// TwinCAT 3 PLC project MyPLC
// ProgramVersion: 3.1.4022.0
// libraries:
//   Tc2_Standard, * (Beckhoff Automation GmbH)
//   Tc2_System, * (Beckhoff Automation GmbH)
//   Tc2_Utilities, * (Beckhoff Automation GmbH)
//   Tc3_Module, * (Beckhoff Automation GmbH)
// project tree:
//   DUTs/Error Monitoring/ ST_HRErrHist.TcDUT
//   DUTs/Signal Generator/ E_DistributionType.TcDUT, E_FunctionType.TcDUT
//   GVLs/ GVL_Constant.TcGVL, GVL_LabviewDataShare.TcGVL
//   / PlcTask.TcTTO
//   POUs/Error Monitoring/ FB_HRErrHist.TcPOU
//   POUs/Signal Generator/ FB_FunctionGenerator.TcPOU (not stored), FB_NoiseGenerator.TcPOU
//   POUs/ MAIN.TcPOU
// real-time tasks:
//   TASK GetDataTask: cycle T#5ms, priority 6, ADS port 350

CONFIGURATION MyPLC
    RESOURCE PLC ON TwinCAT3
        TASK PlcTask(INTERVAL := T#5ms, PRIORITY := 6);
        PROGRAM MAIN WITH PlcTask : MAIN;
    END_RESOURCE
END_CONFIGURATION

// ---- DUTs/Error Monitoring/ST_HRErrHist.TcDUT
TYPE ST_HRErrHist :
STRUCT
{attribute 'displaymode':='hex'}
	hrErrCode	: HRESULT;
	sErrSource	: STRING(63);
	nErrCount	: UDINT;
END_STRUCT
END_TYPE

// ---- DUTs/Signal Generator/E_DistributionType.TcDUT
{attribute 'qualified_only'}
TYPE E_DistributionType :
(
	Uniform := 0,
	Normal,
	Chi_squared,
	Exponential,
	Gamma
);
END_TYPE

// ---- DUTs/Signal Generator/E_FunctionType.TcDUT
{attribute 'qualified_only'}
TYPE E_FunctionType :
(
	Sine,		// typical for vibrations originating from rotating machine
	Square,		// mixed sine signals good for analyzing spectrum
	Pulse,		// mixed sine signals good for analyzing spectrum
	Triangular,	// mixed sine signals good for analyzing spectrum
	Sawtooth,	// ramp-type vibrations, continuously increasing
	AM			// amplitude modulation: typical for vibrations originating from gear-tooth failure or bearing faults
);
END_TYPE

// ---- GVLs/GVL_Constant.TcGVL
VAR_GLOBAL CONSTANT
	
	// input definition
	cChannels		: UDINT 	:= 4;    // number of input channels
	cOversamples 	: UDINT 	:= 10;	 // oversamples from input terminal
	
	// pupulation for statistical calculations
	cPupulation 	: UDINT     := 6000;	
	
	// Source MultiArray
	cBufferLength : UDINT := 100; 
	
	// wait for cAppendData MultiArrays with cBufferLength Elements before calculating | Elements in total = cPupulation 
	cAppendData     : UDINT := cPupulation/cBufferLength;
	
END_VAR

// ---- GVLs/GVL_LabviewDataShare.TcGVL
{attribute 'qualified_only'}
VAR_GLOBAL
	
	//Cal Station Variables	
	out_bInitializeStartupRoutine : BOOL;
	
	 // Beckhoff to Labview MQTT Info Transfer - Current Sensor DeviceID
    out_strDeviceID_labview : STRING;

    // Beckhoff to Labview MQTT Info Transfer - Current Lot running on the Machine
    out_strLotNo_labview : STRING;

    // Beckhoff to Labview MQTT Info Transfer - 1) Calibration 2) FFT
    out_strTestMode_labview : STRING;

    // Beckhoff to Labview MQTT Info Transfer - Interrupt Signal from Beckhoff to Labview to Abort the Calibration Process
    out_bAbortCalibrationSequence_labview : BOOL;

    // Beckhoff to Labview MQTT Info Transfer - Boolean to Indicate if the current sequence are for Master Parts or not
    out_bMasterSequenceActive_labview : BOOL;

    // Beckhoff to Labview MQTT Info Transfer - Boolean indicating the Beckhoff is Active
    out_bBeckhoffHandshakeBit_labview : BOOL;

    // Beckhoff to Labview MQTT Info Transfer - Boolean to Indicate if the current Sensor is Dual Asic or Single ASIC
    out_bDualAsic_labview : BOOL;

    // Beckhoff to Labview MQTT Info Transfer - This bit is to indicate that machine has been reset and now in starting routine
    out_bInitializeStartupRoutine_labview : BOOL;

    // Beckhoff to Labview MQTT Info Transfer - This bit is to indicate that machine is in reset state routine
    out_bRestLabviewRoutine_labview : BOOL;

    // Labview to Beckhoff MQTT Info Transfer - Asic 1 Serial No.
    in_strAsic1SerialNo_labview : STRING;

    // Labview to Beckhoff MQTT Info Transfer - Boolean Indicating Asic 1 Calibration Status Success or not
    in_bAsic1CalibrationSuccess_labview : BOOL;

    // Labview to Beckhoff MQTT Info Transfer - Boolean indicating Asic 1 Calibration In progress
    in_bAsic1CalibrationInProgress_labview : BOOL;

    // Labview to Beckhoff MQTT Info Transfer - Boolean indicating Asic 1 Calibration completed successfully
    in_bAsic1CalibrationCompleted_labview : BOOL;

    // Labview to Beckhoff MQTT Info Transfer - Asic 2 Serial No.
    in_strAsic2SerialNo_labview : STRING;

    // Labview to Beckhoff MQTT Info Transfer - Boolean Indicating Asic 2 Calibration Status Success or not
    in_bAsic2CalibrationSuccess_labview : BOOL;

    // Labview to Beckhoff MQTT Info Transfer - Boolean indicating Asic 2 Calibration In progress
    in_bAsic2CalibrationInProgress_labview : BOOL;

    // Labview to Beckhoff MQTT Info Transfer - Boolean indicating Asic 2 Calibration completed successfully
    in_bAsic2CalibrationCompleted_labview : BOOL;

    // Labview to Beckhoff MQTT Info Transfer - Boolean Indicating if there is an error in Aardvark Board present in the calibration station
    in_bAardvarkBoardError_labview : BOOL;

    // Labview to Beckhoff MQTT Info Transfer - Boolean indicating if there is an error in PTC04 board present in the Calibration station
    in_bPTC04BoardError_labview : BOOL;

    // Labview to Beckhoff MQTT Info Transfer - Boolean indicating if there is an error in NIDaq board present in the Calibration station
    in_bNIDaqError_labview : BOOL;

    // Labview to Beckhoff MQTT Info Transfer - Boolean indicating the Labview is Active
    in_bLabviewHandshakeBit : BOOL;

    // Labview to Beckhoff MQTT Info Transfer - Boolean indicating that Calibration Results have been sent to Database Successfully
    in_bCalResultsDBStoreSuccess_labview : BOOL;

    // Labview to Beckhoff MQTT Info Transfer - This boolean indicates that Startup Initialization routine is now successful
    in_bStartupInitializationSuccess_labview : BOOL;

    // Labview to Beckhoff MQTT Info Transfer - This boolean indicates that Startup Initialization routine is now completed
    in_bStartupInitializationCompleted_labview : BOOL;

    // Labview to Beckhoff MQTT Info Transfer - This boolean indicates that Reset routine is now completed
    in_bLabviewResetComplete_labview : BOOL;

    // Labview to Beckhoff MQTT Info Transfer - This boolean indicates that Reset routine is now successful
    in_bLabviewResetSuccess_labview : BOOL;
	
	//FFT Variables
	
	 // Beckhoff to Labview MQTT Info Transfer - Current Sensor DeviceID
//    out_strDeviceID_labview: STRING; 

    // Beckhoff to Labview MQTT Info Transfer - Current Lot running on the Machine
//    out_strLotNo_labview: STRING; 

    // Beckhoff to Labview MQTT Info Transfer - 1) Calibration 2) FFT
//    out_strTestMode_labview: STRING; 

    // Beckhoff to Labview MQTT Info Transfer - Interrupt Signal from Beckhoff to Labview to Abort the FFT Process
    out_bAbortFFTSequence_labview: BOOL; 

    // Beckhoff to Labview MQTT Info Transfer - Boolean to Indicate if the current sequence are for Master Parts or not
//    out_bMasterSequenceActive_labview: BOOL; 

    // Beckhoff to Labview MQTT Info Transfer - Boolean indicating the Beckhoff is Active. Labview program relies on this signal to make sure Beckhoff communication is active. If this is false, Labview assumes that Labview-Beckhoff communication failed
//    out_bBeckhoffHandshakeBit_labview: BOOL; 

    // Beckhoff to Labview MQTT Info Transfer - Boolean to Indicate if the current Sensor is Dual Asic or Single ASIC
//    out_bDualAsic_labview: BOOL; 

    // Beckhoff to Labview MQTT Info Transfer - This bit is to indicate that machine has been reset and now in starting routine. Please initialize the labview program and get ready for a next trigger for FFT / characterization.
//    out_bInitializeStartupRoutine_labview: BOOL; 

    // Beckhoff to Labview MQTT Info Transfer - This bit is to indicate that machine is in reset state routine. Please Reset the labview program and get ready for startup routine trigger
//    out_bRestLabviewRoutine_labview: BOOL; 

    // Labview to Beckhoff MQTT Info Transfer - Boolean Indicating Asic 1 FFT Status Success or not
    in_bAsic1FFTSuccess_labview: BOOL; 

    // Labview to Beckhoff MQTT Info Transfer - Boolean indicating Asic 1 FFT In progress
    in_bAsic1FFTInProgress_labview: BOOL; 

    // Labview to Beckhoff MQTT Info Transfer - Boolean indicating Asic 1 FFT completed successfully
    in_bAsic1FFTCompleted_labview: BOOL; 

    // Labview to Beckhoff MQTT Info Transfer - Boolean Indicating Asic 2 FFT Status Success or not
    in_bAsic2FFTSuccess_labview: BOOL; 

    // Labview to Beckhoff MQTT Info Transfer - Boolean indicating Asic 2 FFT In progress
    in_bAsic2FFTInProgress_labview: BOOL; 

    // Labview to Beckhoff MQTT Info Transfer - Boolean indicating Asic 2 FFT completed successfully
    in_bAsic2FFTCompleted_labview: BOOL; 

    // Labview to Beckhoff MQTT Info Transfer - Boolean Indicating if there is an error in Aardvark Board present in the FFT station
//    in_bAardvarkBoardError_labview: BOOL; 

    // Labview to Beckhoff MQTT Info Transfer - Boolean indicating if there is an error in PTC04 board present in the FFT station
//    in_bPTC04BoardError_labview: BOOL; 

    // Labview to Beckhoff MQTT Info Transfer - Boolean indicating if there is an error in NIDaq board present in the FFT station
//    in_bNIDaqError_labview: BOOL; 

    // Labview to Beckhoff MQTT Info Transfer - Boolean indicating the Labview is Active. Beckhoff relies on this signal to make sure labview communication is active. If this is false, Beckhoff assumes that Beckhoff Labview communication failed
//    in_bLabviewHandshakeBit: BOOL; 

    // Labview to Beckhoff MQTT Info Transfer - Boolean indicating that FFT Results have been sent to Database Successfully
    in_bFFTResultsDBStoreSuccess_labview: BOOL; 

    // Labview to Beckhoff MQTT Info Transfer - This boolean indicates that Startup Initialization routine is now successful
//    in_bStartupInitializationSuccess_labview: BOOL; 

    // Labview to Beckhoff MQTT Info Transfer - This boolean indicates that Startup Initialization routine is now completed
//    in_bStartupInitializationCompleted_labview: BOOL; 

    // Labview to Beckhoff MQTT Info Transfer - This boolean indicates that Reset routine is now completed
//    in_bLabviewResetComplete_labview: BOOL; 

    // Labview to Beckhoff MQTT Info Transfer - This boolean indicates that Reset routine is now successful
//    in_bLabviewResetSuccess_labview: BOOL; 
	
	
	
END_VAR

// ---- POUs/MAIN.TcPOU
PROGRAM MAIN

VAR
	fbNoiseGeneratorCh1		: FB_NoiseGenerator;		// Signal Generator
	fbNoiseGeneratorCh2		: FB_NoiseGenerator;		// Signal Generator	
	fbFunctionGeneratorCh3	: FB_FunctionGenerator;		// Sine Signal Generator	
	fbFunctionGeneratorCh4	: FB_FunctionGenerator;		// AM Signal Generator
	fbFunctionGeneratorCh5	: FB_FunctionGenerator;		// Square Signal Generator
	fbFunctionGeneratorCh6	: FB_FunctionGenerator;		// Pulse Signal Generator
	
	aNoise_1 : ARRAY[1..cOversamples] OF LREAL;
	aNoise_2 : ARRAY[1..cOversamples] OF LREAL;
	aSine : ARRAY[1..cOversamples] OF LREAL;
	aAM : ARRAY[1..cOversamples] OF LREAL;
	aSquare : ARRAY[1..cOversamples] OF LREAL;
	aPulse : ARRAY[1..cOversamples] OF LREAL;
	
	nStartSeed		: INT := 1;	
	aNormDisp		: ARRAY [1..2] OF LREAL := [1,3];	// mean = 1, std = 3
	aGammaDisp      : ARRAY [1..2] OF LREAL := [4,0];   // DOF = 4
	fSetFrequency	: LREAL := 40;						// Hz
	fSetAmplitude	: LREAL := 10;						// peak amplitude of sine signal
		
END_VAR

// Generate test signals
// Ch1: Normal distribution
// Ch2: Gamma distribution
// Ch3: Sine signal
// Ch4: Triangular signal
fbNoiseGeneratorCh1(	nSeed 		:= nStartSeed,
						aParam 		:= aNormDisp,
						eDistrType	:= E_DistributionType.Normal,								
						aSignal		:= aNoise_1 );	
fbNoiseGeneratorCh2(	nSeed 		:= nStartSeed,
						aParam 		:= aGammaDisp,
						eDistrType	:= E_DistributionType.Gamma,								
						aSignal		:= aNoise_2 );									
fbFunctionGeneratorCh3(	fFrequency 	:= fSetFrequency,
						fAmplitude 	:= fSetAmplitude,
						fOffset		:= 0,
						eFunction 	:= E_FunctionType.Sine,							
						aSignal		:= aSine );
fbFunctionGeneratorCh4(	fFrequency 	:= fSetFrequency,
						fAmplitude 	:= fSetAmplitude,
						fOffset 	:= 0,
						eFunction	:= E_FunctionType.AM,
						aSignal 	:= aAM);
fbFunctionGeneratorCh5(	fFrequency 	:= fSetFrequency,
						fAmplitude 	:= fSetAmplitude,
						fOffset 	:= 0,
						eFunction	:= E_FunctionType.Square,
						aSignal 	:= aSquare);
fbFunctionGeneratorCh6(	fFrequency 	:= fSetFrequency,
						fAmplitude 	:= fSetAmplitude,
						fOffset 	:= 0,
						eFunction	:= E_FunctionType.Pulse,
						aSignal 	:= aPulse);

END_PROGRAM

// ---- POUs/Signal Generator/FB_NoiseGenerator.TcPOU
// generates a random noise signal, typical for disturbance signal. v1.2
// aParam explained
// Uniform 		: aParam[1] := min , aParam[2] := max limit
// Normal	 	: aParam[1] := mean, aParam[2] := standard deviation
// Exponential 	: aParam[1] := mean, aParam[2] := NA
// Gamma		: aParam[1] := deg. of freedom (max. 10), aParam[2] := NA (Gamma distribution: summing DOF number of exp. distributed variables)
// Chi-Squared 	: aParam[1] := mean, aParam[2] := standard deviation (Chi-squared (1DOF) is square of Gaussian Normal)
FUNCTION_BLOCK FB_NoiseGenerator
VAR_INPUT
	bEnable		: BOOL 	:= TRUE;	// set TRUE to generate the specified signal; set FALSE to reset the signal buffer
	nSeed		: INT	:= 1;	 	// seed value (initial value) for random function
	aParam		: ARRAY [1..2] OF LREAL := [0,1];	// specific parameter for chosen distribution type (see FB documentation)
	eDistrType	: E_DistributionType := E_DistributionType.Normal;
END_VAR
VAR_IN_OUT
	aSignal		: ARRAY[1..cOversamples] OF LREAL;
END_VAR
VAR_OUTPUT
	bError		: BOOL;
END_VAR

VAR
	bInit			: BOOL := TRUE;
	nInfiniteValue	: UDINT; // logarithm result is infinite probable caused by a random number of 0.

	nSamples		: UDINT; // array index
	fbRAND			: DRAND;

	// only for Gamma distribution
	nDof			: UINT; // array index
	nMaxDof 		: UINT;		
END_VAR
VAR CONSTANT
	cMaxDofGamma	: UINT := 10;
END_VAR

IF bEnable THEN
	IF bInit THEN
		// Flush out old data
		MEMSET(ADR(aSignal), 0, SIZEOF(aSignal));

		IF cOversamples > 0 THEN		
			fbRAND(Seed := nSeed); // initialize DRAND
			bInit := FALSE;
		ELSE
			bError := TRUE;
		END_IF
	END_IF
	
	// Enable function generator
	IF NOT bError THEN
		// random noise: typical for disturbance signal
		Rand();					
	END_IF
ELSE
	// Flush out old data
	MEMSET(ADR(aSignal), 0, SIZEOF(aSignal));
	
	bInit := TRUE;
	bError := FALSE;
END_IF

METHOD PRIVATE Rand
VAR_INPUT
END_VAR

VAR	
	fX1		: LREAL;
	fX2		: LREAL;
	fY1		: LREAL;
	fLnX1	: LREAL;
	fLength : LREAL;
	fD		: LREAL;
END_VAR
{warning disable C0371}

CASE eDistrType OF	
	E_DistributionType.Uniform:	
		fLength := aParam[2] - aParam[1];
		FOR nSamples := 1 TO cOversamples DO
			fbRAND(Num => fX1);	
			aSignal[nSamples] := fX1 * fLength + aParam[1];
		END_FOR
		
	E_DistributionType.Exponential:		
		FOR nSamples := 1 TO cOversamples DO
			fbRAND(Num => fX1);
			IF fX1 = 0 THEN
				fbRAND(Num => fX1);
			END_IF
			fLnX1 := LN(fX1);
			IF LrealIsFinite(fLnX1) THEN			
				aSignal[nSamples] := -aParam[1] * fLnX1;
			ELSE
				nInfiniteValue := nInfiniteValue + 1;
				aSignal[nSamples] := aParam[1];
			END_IF		
		END_FOR
		
	E_DistributionType.Normal:	
		FOR nSamples := 1 TO cOversamples DO
			// create 2 uniform distributed variables
			fbRAND(Num => fX1);
			IF fX1 = 0 THEN
				fbRAND(Num => fX1);
			END_IF		
			fbRAND(Num => fX2);
			IF fX2 = 0 THEN
				fbRAND(Num => fX2);
			END_IF	
			// create normal distribution
			fLnX1 := LN(fX1);
			IF LrealIsFinite(fLnX1) THEN			
				IF (fLnX1 < 0) THEN
					// Box Müller method
					fY1 := SQRT(-2*fLnX1)*COS(2*PI*fX2);
//					fY2 := SQRT(-2*LN(fX1))*SIN(2*PI*fX2);	
				END_IF
				aSignal[nSamples] := aParam[1] + aParam[2]*fY1;
			ELSE
				nInfiniteValue := nInfiniteValue + 1;
				aSignal[nSamples] := aParam[1];
			END_IF
		END_FOR	
	
	E_DistributionType.Gamma:		
		IF LREAL_TO_UINT(aParam[1]) > cMaxDofGamma THEN
			nMaxDof := cMaxDofGamma;
		ELSE
			nMaxDof := LREAL_TO_UINT(aParam[1]);
		END_IF
		//		
		FOR nSamples := 1 TO cOversamples DO
			aSignal[nSamples] := 0;
			FOR nDof := 1 TO nMaxDof DO
				fbRAND(Num => fX1);
				IF fX1 = 0 THEN
					fbRAND(Num => fX1);
				END_IF
				fLnX1 := LN(fX1);
				IF LrealIsFinite(fLnX1) THEN
					aSignal[nSamples] := aSignal[nSamples] - fLnX1;
				ELSE
					nInfiniteValue := nInfiniteValue + 1;
				END_IF		
			END_FOR	
		END_FOR

	//  1DOF: square of a single gaussian normal variable
	E_DistributionType.Chi_squared:
		FOR nSamples := 1 TO cOversamples DO
			// create 2 uniform distributed variables
			fbRAND(Num => fX1);
			IF fX1 = 0 THEN
				fbRAND(Num => fX1);
			END_IF	
			fbRAND(Num => fX2);
			IF fX2 = 0 THEN
				fbRAND(Num => fX2);
			END_IF	
			// create normal distribution
			fLnX1 := LN(fX1);
			IF LrealIsFinite(fLnX1) THEN				
				IF (fLnX1 < 0) THEN
					// Box Müller method
					fY1 := SQRT(-2*fLnX1)*COS(2*PI*fX2);
//					fY2 := SQRT(-2*LN(fX1))*SIN(2*PI*fX2);	
				END_IF	
				fD := aParam[1] + aParam[2]*fY1;
			ELSE
				nInfiniteValue := nInfiniteValue + 1;
				fD := aParam[1];		
			END_IF
			aSignal[nSamples] := fD * fD;
		END_FOR
		
END_CASE

{warning restore C0371}
END_METHOD

END_FUNCTION_BLOCK

// ---- POUs/Error Monitoring/FB_HRErrHist.TcPOU
FUNCTION_BLOCK FB_HRErrHist
(* v1.10
build up an error history consisting of two arrays and one index.
The index shows the actual array position. The last error id and the count for this id are saved in the arrays.
If an error id is the same as the previous input error the counter is increased. Otherwise the index is increased.
*)
VAR_INPUT
	bEdgeDetect	: BOOL;	(* FALSE: every input(bErr) is processed; TRUE: only rising edge of input is processed *)
END_VAR
VAR_OUTPUT
	nErrSum		: UINT;
	nErrIdx		: UINT; // error list index of last occured error (max. cHistLen)
	aErrList	: ARRAY[1..cHistLen] OF ST_HRErrHist;
END_VAR

VAR
	bNewErr		: BOOL;
	fbErrTrig	: R_TRIG;
END_VAR
VAR CONSTANT
	cHistLen	: UINT := 100;
END_VAR

METHOD AddError
VAR_INPUT
	bErr		: BOOL;
	hrErrCode	: HRESULT;
	sErrSource	: STRING(63);
END_VAR
fbErrTrig(CLK:=bErr);
IF bEdgeDetect THEN
	bNewErr := fbErrTrig.Q;
ELSE
	bNewErr := bErr;
END_IF

IF bNewErr THEN
	nErrSum := nErrSum + 1;
	IF nErrIdx < cHistLen THEN
		IF nErrIdx = 0 THEN
			nErrIdx	:= nErrIdx + 1;
		ELSIF aErrList[nErrIdx].hrErrCode <> hrErrCode OR aErrList[nErrIdx].sErrSource <> sErrSource THEN
			nErrIdx	:= nErrIdx + 1;
		END_IF
		aErrList[nErrIdx].hrErrCode := hrErrCode;
		aErrList[nErrIdx].sErrSource := sErrSource;
		aErrList[nErrIdx].nErrCount := aErrList[nErrIdx].nErrCount + 1;
	END_IF
END_IF
END_METHOD

METHOD Reset
VAR_INPUT
END_VAR
nErrSum := 0;
nErrIdx := 0;
MEMSET(ADR(aErrList),0,SIZEOF(aErrList));
END_METHOD

END_FUNCTION_BLOCK
